{attribute 'enable_dynamic_creation'}
{attribute 'no_explicit_call' := 'Do not call the body - Stick to OOP'}
FUNCTION_BLOCK FB_XP_Path EXTENDS FB_CH_Object IMPLEMENTS I_XP_Path
VAR
	fbTracksUsed : FB_CH_List;
	ipStartStation, ipDestinationStation : I_XP_Station;
	fPathLength : LREAL;
END_VAR

METHOD DistanceToDestiantion : LREAL
VAR_INPUT
	ipTrack : I_XP_Track;
	fPosOnTrack : LREAL;
END_VAR
VAR
	bCorrectPos, bCorrectTrack : BOOL;
	bPosFound : BOOL;
	fDistReturnNotOnThisTrack : LREAL;
	fStart, fEnd : LREAL;
	ipEachTrack : I_XP_Track; 
END_VAR
VAR
	//Todo add tolerance to Size >1
	fToleranceWindow : LREAL := 0.001;//[mm] if Mover is this distance mor far away from the parent, return 0mm
END_VAR
IF ipTrack = 0 THEN
	//Error -  invalide interface
	DistanceToDestiantion := CHALET_BaseComponents.GVL_Datatypes.cMaxLreal;
	RETURN;
END_IF

fDistReturnNotOnThisTrack := CHALET_BaseComponents.GVL_Datatypes.cMaxLreal;

IF (fbTracksUsed.OIDInList(ipTrack.OID) = 0) OR fPosOnTrack < 0 OR  fPosOnTrack > ipTrack.Length THEN
	//Error -  position not on track
	DistanceToDestiantion := fDistReturnNotOnThisTrack;
	RETURN;
END_IF


IF fbTracksUsed.Size = 1 THEN
	bCorrectPos := F_InLimitTest(fMinimum :=  THIS^.StationStart.PositionOnTrack, fInput:=fPosOnTrack , fMaximum:=  (THIS^.StationDestination.PositionOnTrack + fToleranceWindow));
	bCorrectTrack := (ipTrack = StationDestination.AccocietedTrack);

	IF bCorrectPos AND bCorrectTrack THEN
		DistanceToDestiantion := F_GetDistToPosModulo(fTargetPosition := THIS^.StationDestination.PositionOnTrack, fActualPosition := fPosOnTrack, fModulo := ipTrack.Length);
		//check tolerance window
		IF (DistanceToDestiantion + fToleranceWindow) >= ipTrack.Length THEN
			DistanceToDestiantion := 0.0;
		END_IF
	ELSE
		DistanceToDestiantion := fDistReturnNotOnThisTrack;
	END_IF
	RETURN;
END_IF


IF fbTracksUsed.Size > 1 THEN 
	fbTracksUsed.ResetIterator();	
	
	////First track in list
	IF ToXpTrack(fbTracksUsed.GetNextObject(),ipEachTrack) THEN
		fStart 	:= THIS^.StationStart.PositionOnTrack;
		fEnd 	:= ipEachTrack.Length;
		
		bCorrectPos := F_InLimitTest(fMinimum :=  fStart, fInput:=fPosOnTrack , fMaximum:=  fEnd);
		bCorrectTrack := (ipTrack = ipEachTrack);
		IF bCorrectPos AND bCorrectTrack THEN
			bPosFound := TRUE;
			DistanceToDestiantion := fEnd - fPosOnTrack;
		END_IF
	END_IF
	
	
	//All tracks in between
	WHILE fbTracksUsed.HasNextObject() DO
		IF ToXpTrack(fbTracksUsed.GetNextObject(),ipEachTrack) AND_THEN fbTracksUsed.HasNextObject() THEN
			fStart 	:= 0;
			fEnd 	:= ipEachTrack.Length;
			
			// still locking for the startpoint to measure the distance to Destination
			IF NOT bPosFound THEN
				bCorrectPos := F_InLimitTest(fMinimum :=  fStart, fInput:=fPosOnTrack , fMaximum:=  fEnd);
				bCorrectTrack := (ipTrack = ipEachTrack);
				IF bCorrectPos AND bCorrectTrack THEN
					bPosFound := TRUE;
					DistanceToDestiantion := fEnd - fPosOnTrack;
				END_IF
			ELSE
				// add all the tracklengths
				DistanceToDestiantion := DistanceToDestiantion + fEnd;		
			END_IF
		END_IF
	END_WHILE	
	
	
	//Last track
		fStart 	:= 0;
		fEnd 	:= (THIS^.StationDestination.PositionOnTrack + fToleranceWindow);
		// still locking for the startpoint to measure the distance to Destination
		IF NOT bPosFound THEN
			bCorrectPos := F_InLimitTest(fMinimum :=  fStart, fInput:=fPosOnTrack , fMaximum :=  fEnd);
			bCorrectTrack := (ipTrack = ipEachTrack);
			IF bCorrectPos AND bCorrectTrack THEN
				bPosFound := TRUE;
				DistanceToDestiantion := MAX(0, THIS^.StationDestination.PositionOnTrack - fPosOnTrack);
			END_IF
		ELSE
			// add all the tracklengths
			DistanceToDestiantion := DistanceToDestiantion + fEnd;		
		END_IF

	
	fbTracksUsed.RestoreIterator();
	
	IF NOT bPosFound THEN
		DistanceToDestiantion := fDistReturnNotOnThisTrack;
		RETURN;
	END_IF
END_IF
END_METHOD

{attribute 'monitoring':='call'}
//[mm]
PROPERTY Length : LREAL
GET
Length := THIS^.fPathLength;
END_GET
SET
THIS^.fPathLength := Length;
END_SET
END_PROPERTY

{attribute 'monitoring':='call'}
PROPERTY LUID : STRING //Locally unique identifier
GET
VAR
	sTempName : STRING;
END_VAR
IF ipStartStation <> 0 AND ipDestinationStation <> 0 THEN
	sTempName := CONCAT(sTempName, ipStartStation.LUID);
	sTempName := CONCAT(sTempName, ' to ' );
	sTempName := CONCAT(sTempName, ipDestinationStation.LUID);
	
ELSIF ipStartStation <> 0 THEN
	sTempName := CONCAT(sTempName, ipStartStation.LUID);
	sTempName := CONCAT(sTempName, ' to ?' );

ELSIF ipDestinationStation <> 0 THEN
	sTempName := CONCAT(sTempName, '? to ' );
	sTempName := CONCAT(sTempName, ipDestinationStation.LUID);
	
ELSE 
	sTempName := ' Unknown path';
END_IF


LUID := sTempName;
END_GET
END_PROPERTY

{attribute 'monitoring':='call'}
PROPERTY StationDestination : I_XP_Station
GET
StationDestination := THIS^.ipDestinationStation;
END_GET
SET
THIS^.ipDestinationStation := StationDestination;
END_SET
END_PROPERTY

{attribute 'monitoring':='call'}
PROPERTY StationStart  : I_XP_Station
GET
StationStart := THIS^.ipStartStation;
END_GET
SET
THIS^.ipStartStation := StationStart;
END_SET
END_PROPERTY

{attribute 'monitoring':='call'}
//List of tracks
PROPERTY TracksUsed : REFERENCE TO FB_CH_List
GET
TracksUsed REF= THIS^.fbTracksUsed;
END_GET
END_PROPERTY

END_FUNCTION_BLOCK

(* stored: Version 1.1.0.1, ProductVersion 3.1.4024.15
   POU FB_XP_Path: Id {a479f742-a551-40e5-a493-f32ce50e69f9}, SpecialFunc None
   Method DistanceToDestiantion: Id {49fa156c-c599-49f7-8c5b-c2e0b1d7c185}
   Property Length: Id {9957ab4a-c60a-4dda-8b93-f3628e87faf2}
   Get Get: Id {200d8c22-a772-4dfe-ac22-68adb8102b4c}
   Set Set: Id {da0da2b0-41d5-4c9d-ab98-d16d71e56be3}
   Property LUID: Id {26d11d55-a790-4b46-8b31-b39f504198af}
   Get Get: Id {e088ce95-219f-484b-a793-c4a4c26a3f58}
   Property StationDestination: Id {1b455b3b-bd79-486d-9910-39e95da55283}
   Get Get: Id {e8310971-86a0-43ac-9a0f-6b8c4a2bb8ad}
   Set Set: Id {8358497b-03af-4ad4-a8b3-32fd9425ecfd}
   Property StationStart: Id {22f96e9a-bf89-4243-809d-d2d258473025}
   Get Get: Id {f3060c35-9b14-48ce-8c37-20e0c7535eaa}
   Set Set: Id {e84cf6fc-7f5b-48ae-8af3-01d8c941bb25}
   Property TracksUsed: Id {5170e2b5-479c-4450-80bf-4959ba6b1bca}
   Get Get: Id {cf560e5a-4d4f-4c60-a8c0-e624ca89ff50} *)
